# EPICS substitutions: R1.8.0/edtApp/Db/pluginBldSpectrometer.substitutions
#
# pluginBldSpectrometer db substitutions file
#

file NDPluginBase.template
{
	{
	P=$(CAM):,
	R=BLD$(N):,
	PORT=BLD$(N),
	ADDR=0,
	TIMEOUT=1,
	NDARRAY_PORT=$(PLUGIN_SRC),
	NDARRAY_ADDR=0,
	BIT_DEPTH=$(IMAGE_BIT_DEPTH),
	}
}

file pluginBldSpectrometer.template
{
	{
	P=$(CAM):,
	R=BLD$(N):,
	PORT=BLD$(N),
	HIST_SIZE=256,
	NCHANS=2048,
	ADDR=0,
	TIMEOUT=1
	}
}
